{attribute 'GeneratedUsingTerminal: '}
{attribute addProperty BoxType ""}
{attribute addProperty Id ""}
{attribute addProperty CRC "0"}
{attribute addProperty Size "0"}
TYPE EtcSlaveTerminalBase :
STRUCT
END_STRUCT
END_TYPE

(* stored: Version 1.2.0.0, ProductVersion 3.1.4024.9
   DUT EtcSlaveTerminalBase: Id {4ad0f64e-8eab-4347-b7db-c934e6645e04} *)
